{attribute 'qualified_only'}
{attribute 'strict'}
{attribute 'to_string'}
TYPE E_INSTANCE_CHECK :
(
  NULL,

	POINTER_COLLECTOR_ITF_INVALID := 9000,
  INVALID_INSTANCE_CONTROL_REFERENCE,
  INVALID_INSTANCE_STATE_REFERENCE,
  PROCESS_ID_ZERO := 9100,
  PROCESS_ID_MAX  := 9200,
  PROCESS_ID_NOTEQUAL_COLLECTOR_ID := 9300,
  PROCESS_LIST_ITF_INDEX_INVALID := 9400,

  CHECK_DONE := 10000
)UINT;
END_TYPE

(* stored: Version 1.1.0.1, ProductVersion 3.1.4026.18
   DUT E_INSTANCE_CHECK: Id {7bde2c79-c596-44df-89f1-8d572ca1f76a} *)
